// Mitsubishi GX Works2 project: R3R4R5 plc 20-08-2023_fr   PLC: Q03UDV

PROGRAM MAIN
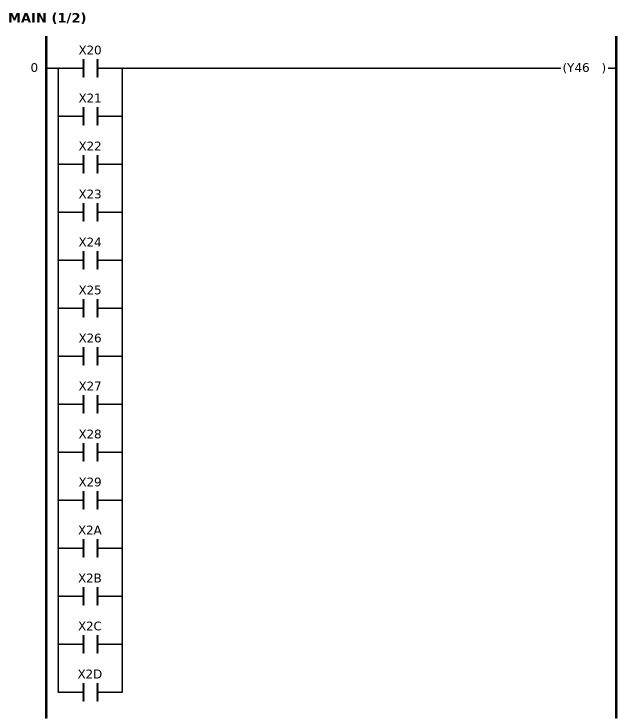
0     LD      X20
      OR      X21
      OR      X22
      OR      X23
      OR      X24
      OR      X25
      OR      X26
      OR      X27
      OR      X28
      OR      X29
      OR      X2A
      OR      X2B
      OR      X2C
      OR      X2D
      OUT     Y46
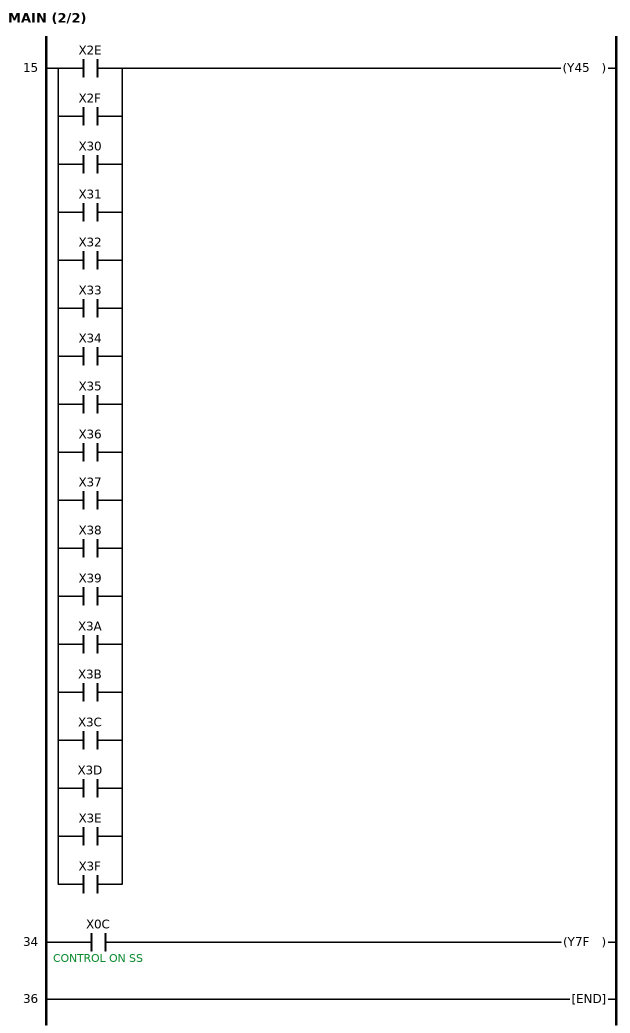
15    LD      X2E
      OR      X2F
      OR      X30
      OR      X31
      OR      X32
      OR      X33
      OR      X34
      OR      X35
      OR      X36
      OR      X37
      OR      X38
      OR      X39
      OR      X3A
      OR      X3B
      OR      X3C
      OR      X3D
      OR      X3E
      OR      X3F
      OUT     Y45
34    LD      X0C  ; CONTROL ON SS
      OUT     Y7F
36    END
END_PROGRAM

PROGRAM DEVICNET
0     END
END_PROGRAM

PROGRAM AUTO_PRG
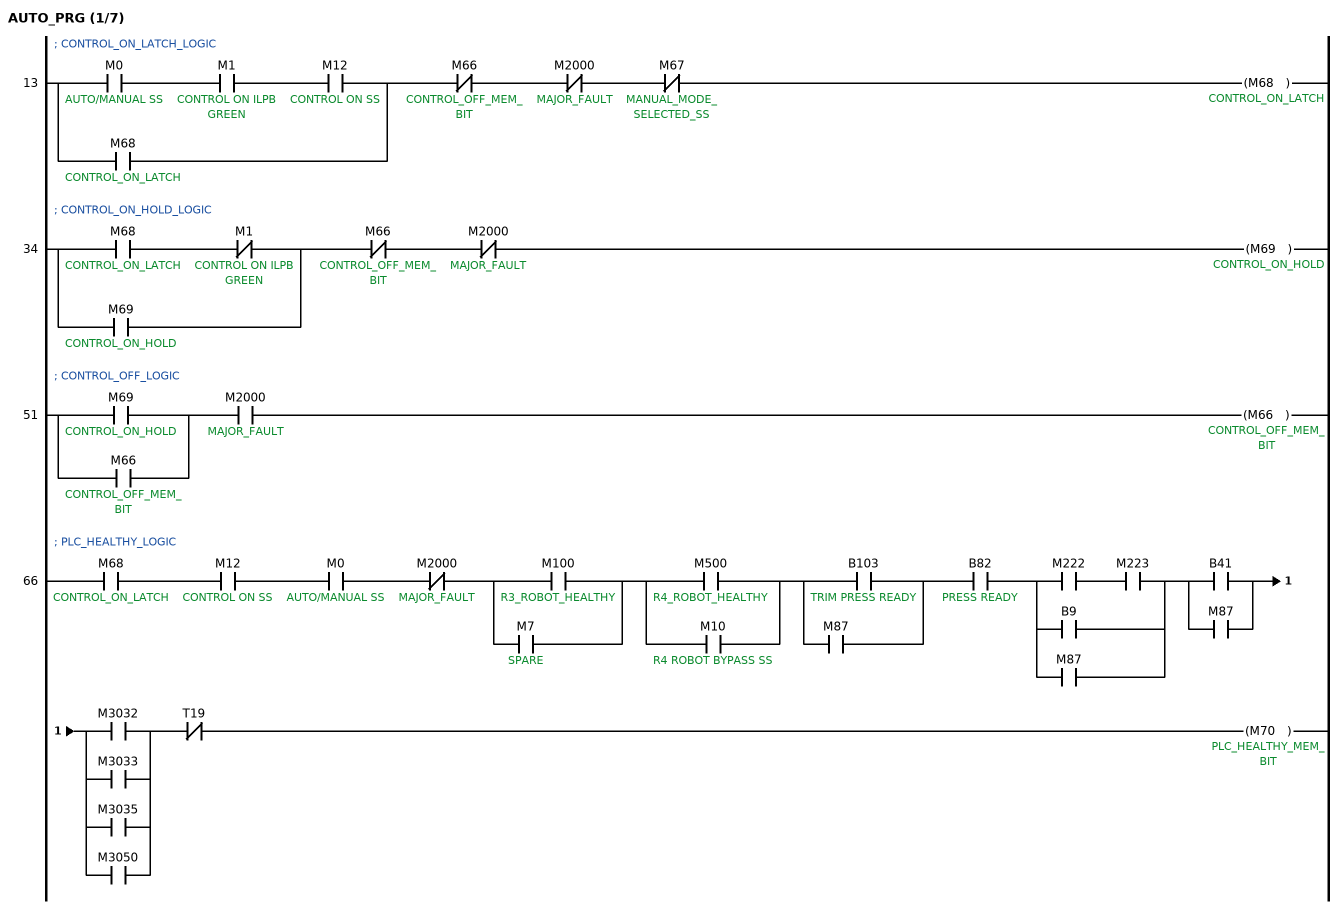
; CONTROL_ON_LATCH_LOGIC
13    LD      M0  ; AUTO/MANUAL SS
      AND     M1  ; CONTROL ON ILPB GREEN
      AND     M12  ; CONTROL ON SS
      OR      M68  ; CONTROL_ON_LATCH
      ANI     M66  ; CONTROL_OFF_MEM_BIT
      ANI     M2000  ; MAJOR_FAULT
      ANI     M67  ; MANUAL_MODE_SELECTED_SS
      OUT     M68  ; CONTROL_ON_LATCH
; CONTROL_ON_HOLD_LOGIC
34    LD      M68  ; CONTROL_ON_LATCH
      ANI     M1  ; CONTROL ON ILPB GREEN
      OR      M69  ; CONTROL_ON_HOLD
      ANI     M66  ; CONTROL_OFF_MEM_BIT
      ANI     M2000  ; MAJOR_FAULT
      OUT     M69  ; CONTROL_ON_HOLD
; CONTROL_OFF_LOGIC
51    LD      M69  ; CONTROL_ON_HOLD
      OR      M66  ; CONTROL_OFF_MEM_BIT
      AND     M2000  ; MAJOR_FAULT
      OUT     M66  ; CONTROL_OFF_MEM_BIT
; PLC_HEALTHY_LOGIC
66    LD      M68  ; CONTROL_ON_LATCH
      AND     M12  ; CONTROL ON SS
      AND     M0  ; AUTO/MANUAL SS
      ANI     M2000  ; MAJOR_FAULT
      LD      M100  ; R3_ROBOT_HEALTHY
      OR      M7  ; SPARE
      ANB
      LD      M500  ; R4_ROBOT_HEALTHY
      OR      M10  ; R4 ROBOT BYPASS SS
      ANB
      LD      B103  ; TRIM PRESS READY
      OR      M87
      ANB
      AND     B82  ; PRESS READY
      LD      M222
      AND     M223
      OR      B9
      OR      M87
      ANB
      LD      B41
      OR      M87
      ANB
      LD      M3032
      OR      M3033
      OR      M3035
      OR      M3050
      ANB
      ANI     T19
      OUT     M70  ; PLC_HEALTHY_MEM_BIT
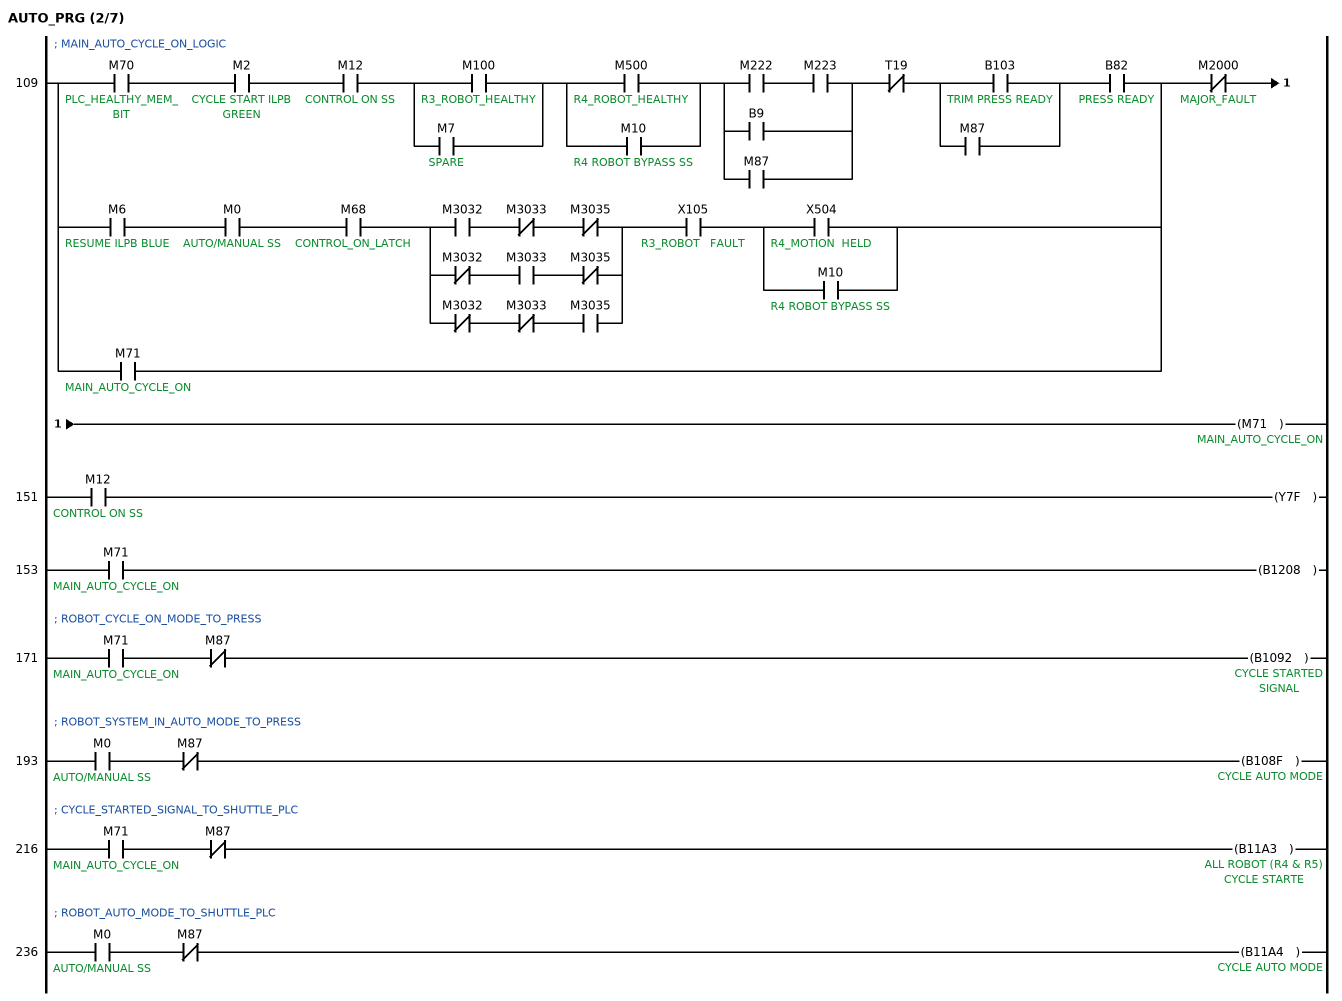
; MAIN_AUTO_CYCLE_ON_LOGIC
109   LD      M70  ; PLC_HEALTHY_MEM_BIT
      AND     M2  ; CYCLE START ILPB GREEN
      AND     M12  ; CONTROL ON SS
      LD      M100  ; R3_ROBOT_HEALTHY
      OR      M7  ; SPARE
      ANB
      LD      M500  ; R4_ROBOT_HEALTHY
      OR      M10  ; R4 ROBOT BYPASS SS
      ANB
      LD      M222
      AND     M223
      OR      B9
      OR      M87
      ANB
      ANI     T19
      LD      B103  ; TRIM PRESS READY
      OR      M87
      ANB
      AND     B82  ; PRESS READY
      LD      M6  ; RESUME ILPB BLUE
      AND     M0  ; AUTO/MANUAL SS
      AND     M68  ; CONTROL_ON_LATCH
      LD      M3032
      ANI     M3033
      ANI     M3035
      LDI     M3032
      AND     M3033
      ANI     M3035
      ORB
      LDI     M3032
      ANI     M3033
      AND     M3035
      ORB
      ANB
      AND     X105  ; R3_ROBOT   FAULT
      LD      X504  ; R4_MOTION  HELD
      OR      M10  ; R4 ROBOT BYPASS SS
      ANB
      ORB
      OR      M71  ; MAIN_AUTO_CYCLE_ON
      ANI     M2000  ; MAJOR_FAULT
      OUT     M71  ; MAIN_AUTO_CYCLE_ON
151   LD      M12  ; CONTROL ON SS
      OUT     Y7F
153   LD      M71  ; MAIN_AUTO_CYCLE_ON
      OUT     B1208
; ROBOT_CYCLE_ON_MODE_TO_PRESS
171   LD      M71  ; MAIN_AUTO_CYCLE_ON
      ANI     M87
      OUT     B1092  ; CYCLE STARTED SIGNAL
; ROBOT_SYSTEM_IN_AUTO_MODE_TO_PRESS
193   LD      M0  ; AUTO/MANUAL SS
      ANI     M87
      OUT     B108F  ; CYCLE AUTO MODE
; CYCLE_STARTED_SIGNAL_TO_SHUTTLE_PLC
216   LD      M71  ; MAIN_AUTO_CYCLE_ON
      ANI     M87
      OUT     B11A3  ; ALL ROBOT (R4 & R5) CYCLE STARTE
; ROBOT_AUTO_MODE_TO_SHUTTLE_PLC
236   LD      M0  ; AUTO/MANUAL SS
      ANI     M87
      OUT     B11A4  ; CYCLE AUTO MODE
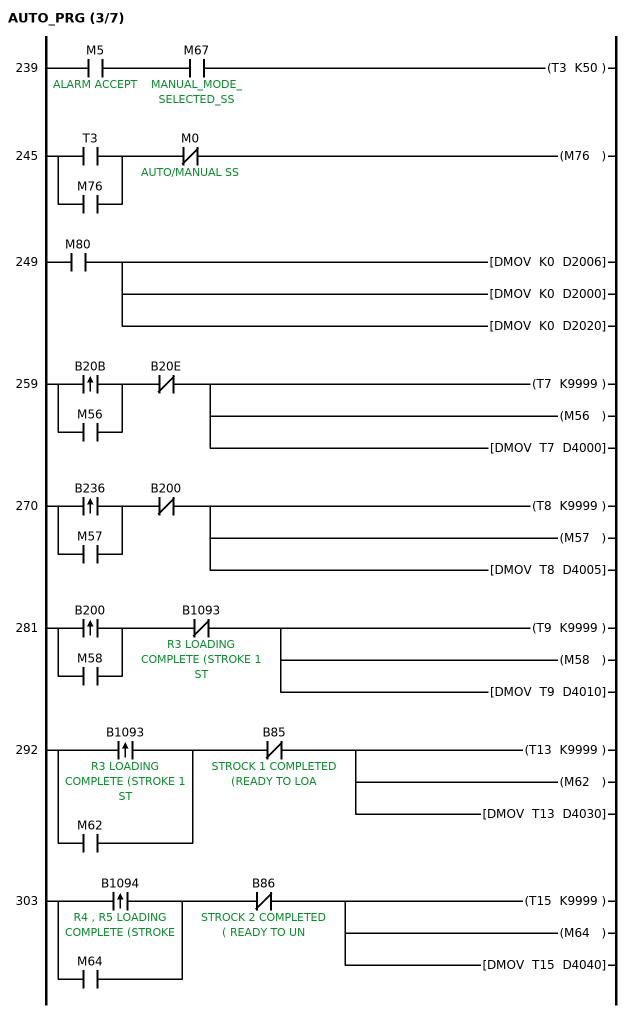
239   LD      M5  ; ALARM ACCEPT
      AND     M67  ; MANUAL_MODE_SELECTED_SS
      OUT     T3 K50
245   LD      T3
      OR      M76
      ANI     M0  ; AUTO/MANUAL SS
      OUT     M76
249   LD      M80
      DMOV    K0 D2006
      DMOV    K0 D2000
      DMOV    K0 D2020
259   LDP     B20B
      OR      M56
      ANI     B20E
      OUT     T7 K9999
      OUT     M56
      DMOV    T7 D4000
270   LDP     B236
      OR      M57
      ANI     B200
      OUT     T8 K9999
      OUT     M57
      DMOV    T8 D4005
281   LDP     B200
      OR      M58
      ANI     B1093  ; R3 LOADING COMPLETE (STROKE 1 ST
      OUT     T9 K9999
      OUT     M58
      DMOV    T9 D4010
292   LDP     B1093  ; R3 LOADING COMPLETE (STROKE 1 ST
      OR      M62
      ANI     B85  ; STROCK 1 COMPLETED (READY TO LOA
      OUT     T13 K9999
      OUT     M62
      DMOV    T13 D4030
303   LDP     B1094  ; R4 , R5 LOADING COMPLETE (STROKE
      OR      M64
      ANI     B86  ; STROCK 2 COMPLETED ( READY TO UN
      OUT     T15 K9999
      OUT     M64
      DMOV    T15 D4040
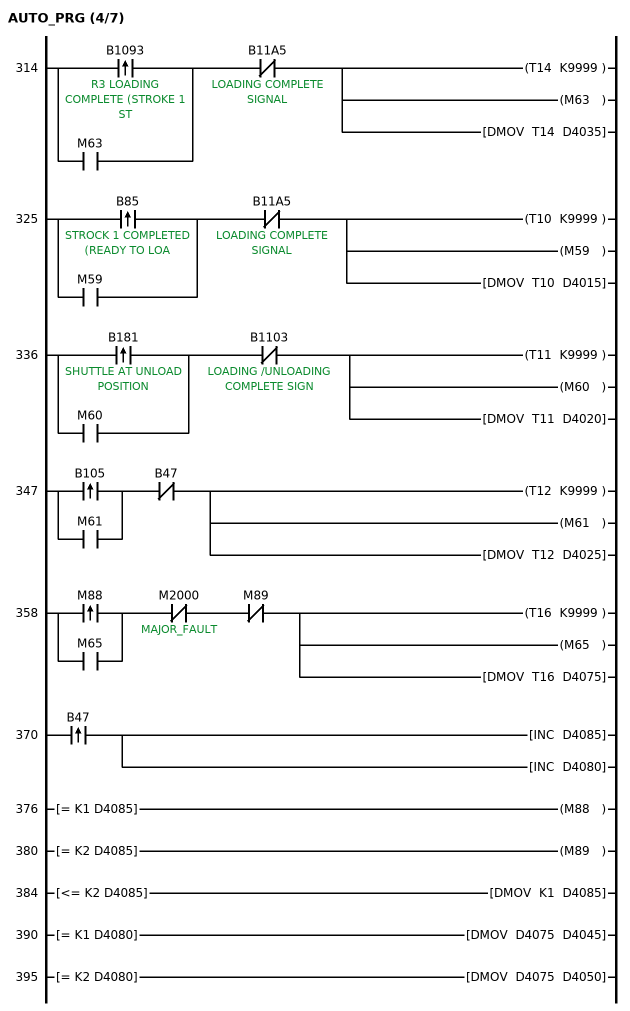
314   LDP     B1093  ; R3 LOADING COMPLETE (STROKE 1 ST
      OR      M63
      ANI     B11A5  ; LOADING COMPLETE SIGNAL
      OUT     T14 K9999
      OUT     M63
      DMOV    T14 D4035
325   LDP     B85  ; STROCK 1 COMPLETED (READY TO LOA
      OR      M59
      ANI     B11A5  ; LOADING COMPLETE SIGNAL
      OUT     T10 K9999
      OUT     M59
      DMOV    T10 D4015
336   LDP     B181  ; SHUTTLE AT UNLOAD POSITION
      OR      M60
      ANI     B1103  ; LOADING /UNLOADING COMPLETE SIGN
      OUT     T11 K9999
      OUT     M60
      DMOV    T11 D4020
347   LDP     B105
      OR      M61
      ANI     B47
      OUT     T12 K9999
      OUT     M61
      DMOV    T12 D4025
358   LDP     M88
      OR      M65
      ANI     M2000  ; MAJOR_FAULT
      ANI     M89
      OUT     T16 K9999
      OUT     M65
      DMOV    T16 D4075
370   LDP     B47
      INC     D4085
      INC     D4080
376   LD=     K1 D4085
      OUT     M88
380   LD=     K2 D4085
      OUT     M89
384   LD<=    K2 D4085
      DMOV    K1 D4085
390   LD=     K1 D4080
      DMOV    D4075 D4045
395   LD=     K2 D4080
      DMOV    D4075 D4050
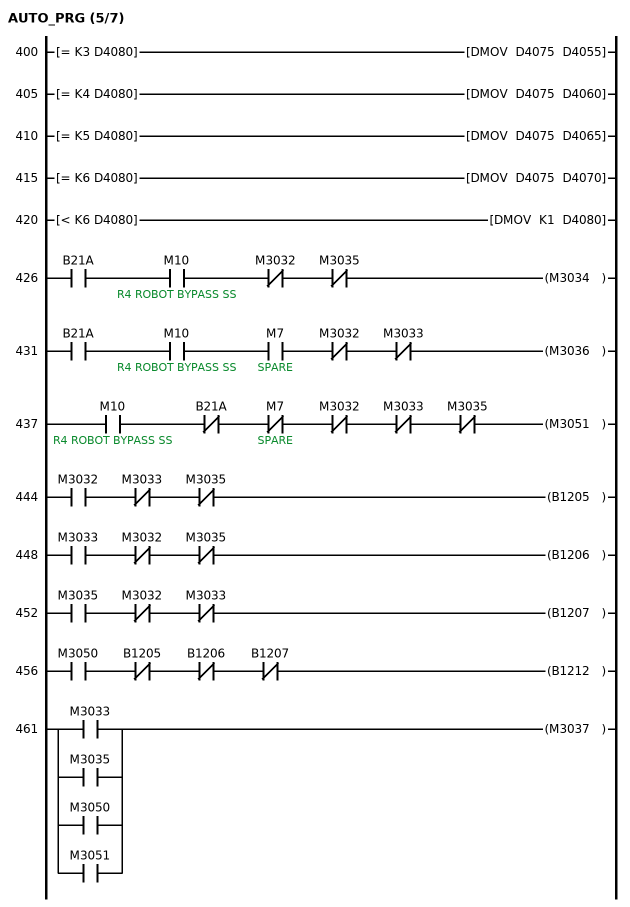
400   LD=     K3 D4080
      DMOV    D4075 D4055
405   LD=     K4 D4080
      DMOV    D4075 D4060
410   LD=     K5 D4080
      DMOV    D4075 D4065
415   LD=     K6 D4080
      DMOV    D4075 D4070
420   LD<     K6 D4080
      DMOV    K1 D4080
426   LD      B21A
      AND     M10  ; R4 ROBOT BYPASS SS
      ANI     M3032
      ANI     M3035
      OUT     M3034
431   LD      B21A
      AND     M10  ; R4 ROBOT BYPASS SS
      AND     M7  ; SPARE
      ANI     M3032
      ANI     M3033
      OUT     M3036
437   LD      M10  ; R4 ROBOT BYPASS SS
      ANI     B21A
      ANI     M7  ; SPARE
      ANI     M3032
      ANI     M3033
      ANI     M3035
      OUT     M3051
444   LD      M3032
      ANI     M3033
      ANI     M3035
      OUT     B1205
448   LD      M3033
      ANI     M3032
      ANI     M3035
      OUT     B1206
452   LD      M3035
      ANI     M3032
      ANI     M3033
      OUT     B1207
456   LD      M3050
      ANI     B1205
      ANI     B1206
      ANI     B1207
      OUT     B1212
461   LD      M3033
      OR      M3035
      OR      M3050
      OR      M3051
      OUT     M3037
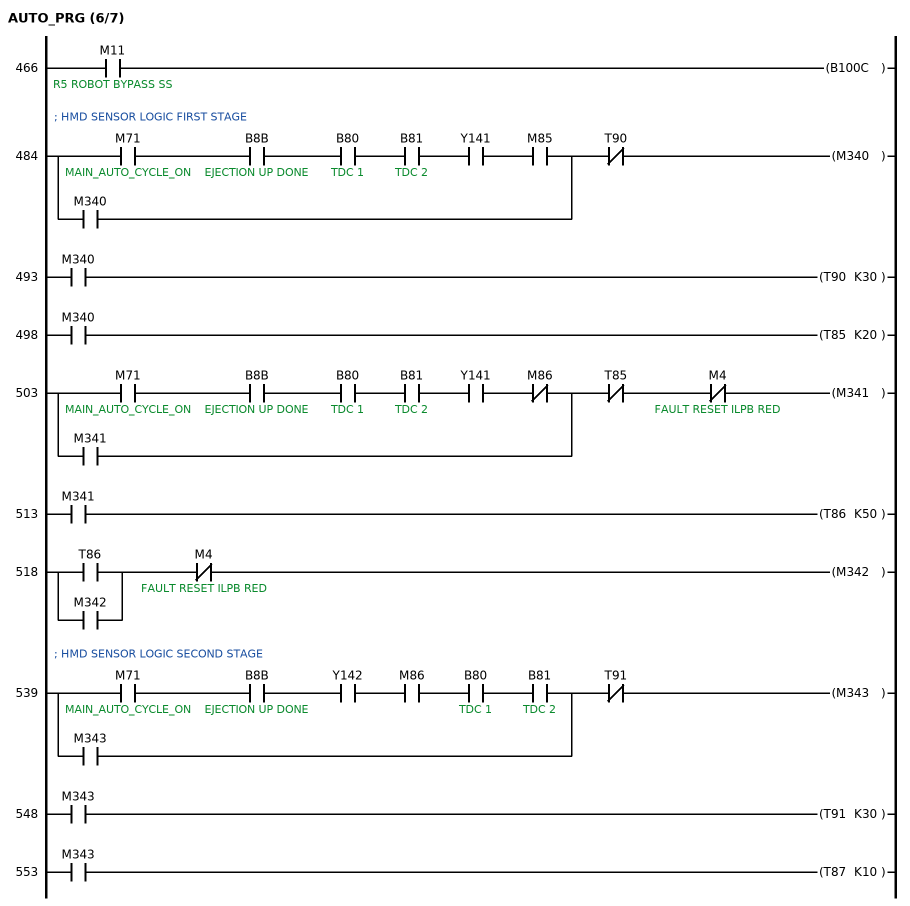
466   LD      M11  ; R5 ROBOT BYPASS SS
      OUT     B100C
; HMD SENSOR LOGIC FIRST STAGE
484   LD      M71  ; MAIN_AUTO_CYCLE_ON
      AND     B8B  ; EJECTION UP DONE
      AND     B80  ; TDC 1
      AND     B81  ; TDC 2
      AND     Y141
      AND     M85
      OR      M340
      ANI     T90
      OUT     M340
493   LD      M340
      OUT     T90 K30
498   LD      M340
      OUT     T85 K20
503   LD      M71  ; MAIN_AUTO_CYCLE_ON
      AND     B8B  ; EJECTION UP DONE
      AND     B80  ; TDC 1
      AND     B81  ; TDC 2
      AND     Y141
      ANI     M86
      OR      M341
      ANI     T85
      ANI     M4  ; FAULT RESET ILPB RED
      OUT     M341
513   LD      M341
      OUT     T86 K50
518   LD      T86
      OR      M342
      ANI     M4  ; FAULT RESET ILPB RED
      OUT     M342
; HMD SENSOR LOGIC SECOND STAGE
539   LD      M71  ; MAIN_AUTO_CYCLE_ON
      AND     B8B  ; EJECTION UP DONE
      AND     Y142
      AND     M86
      AND     B80  ; TDC 1
      AND     B81  ; TDC 2
      OR      M343
      ANI     T91
      OUT     M343
548   LD      M343
      OUT     T91 K30
553   LD      M343
      OUT     T87 K10
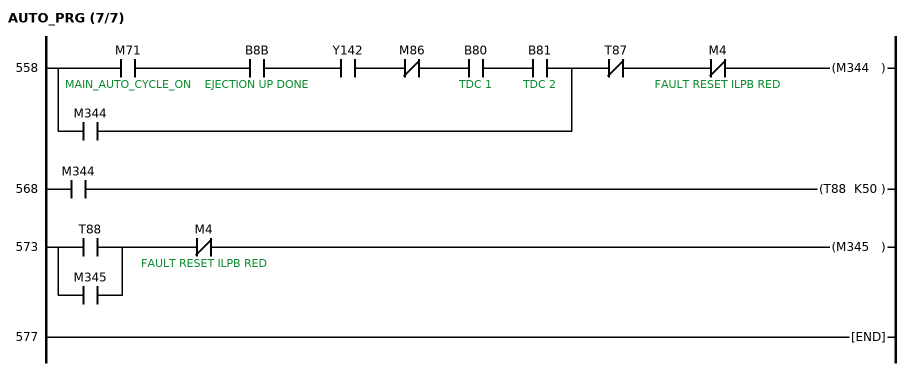
558   LD      M71  ; MAIN_AUTO_CYCLE_ON
      AND     B8B  ; EJECTION UP DONE
      AND     Y142
      ANI     M86
      AND     B80  ; TDC 1
      AND     B81  ; TDC 2
      OR      M344
      ANI     T87
      ANI     M4  ; FAULT RESET ILPB RED
      OUT     M344
568   LD      M344
      OUT     T88 K50
573   LD      T88
      OR      M345
      ANI     M4  ; FAULT RESET ILPB RED
      OUT     M345
577   END
END_PROGRAM

PROGRAM CC_LINK
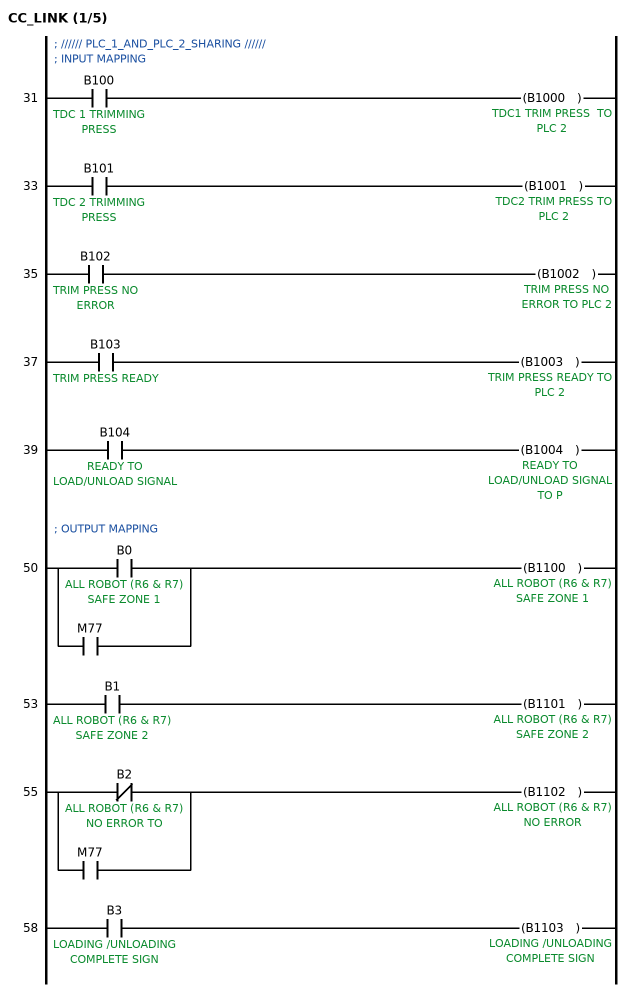
; ////// PLC_1_AND_PLC_2_SHARING //////
; 
; INPUT MAPPING
31    LD      B100  ; TDC 1 TRIMMING PRESS
      OUT     B1000  ; TDC1 TRIM PRESS  TO PLC 2
33    LD      B101  ; TDC 2 TRIMMING PRESS
      OUT     B1001  ; TDC2 TRIM PRESS TO PLC 2
35    LD      B102  ; TRIM PRESS NO ERROR
      OUT     B1002  ; TRIM PRESS NO ERROR TO PLC 2
37    LD      B103  ; TRIM PRESS READY
      OUT     B1003  ; TRIM PRESS READY TO PLC 2
39    LD      B104  ; READY TO LOAD/UNLOAD SIGNAL
      OUT     B1004  ; READY TO LOAD/UNLOAD SIGNAL TO P
; OUTPUT MAPPING
50    LD      B0  ; ALL ROBOT (R6 & R7) SAFE ZONE 1
      OR      M77
      OUT     B1100  ; ALL ROBOT (R6 & R7) SAFE ZONE 1
53    LD      B1  ; ALL ROBOT (R6 & R7) SAFE ZONE 2
      OUT     B1101  ; ALL ROBOT (R6 & R7) SAFE ZONE 2
55    LDI     B2  ; ALL ROBOT (R6 & R7) NO ERROR TO
      OR      M77
      OUT     B1102  ; ALL ROBOT (R6 & R7) NO ERROR
58    LD      B3  ; LOADING /UNLOADING COMPLETE SIGN
      OUT     B1103  ; LOADING /UNLOADING COMPLETE SIGN
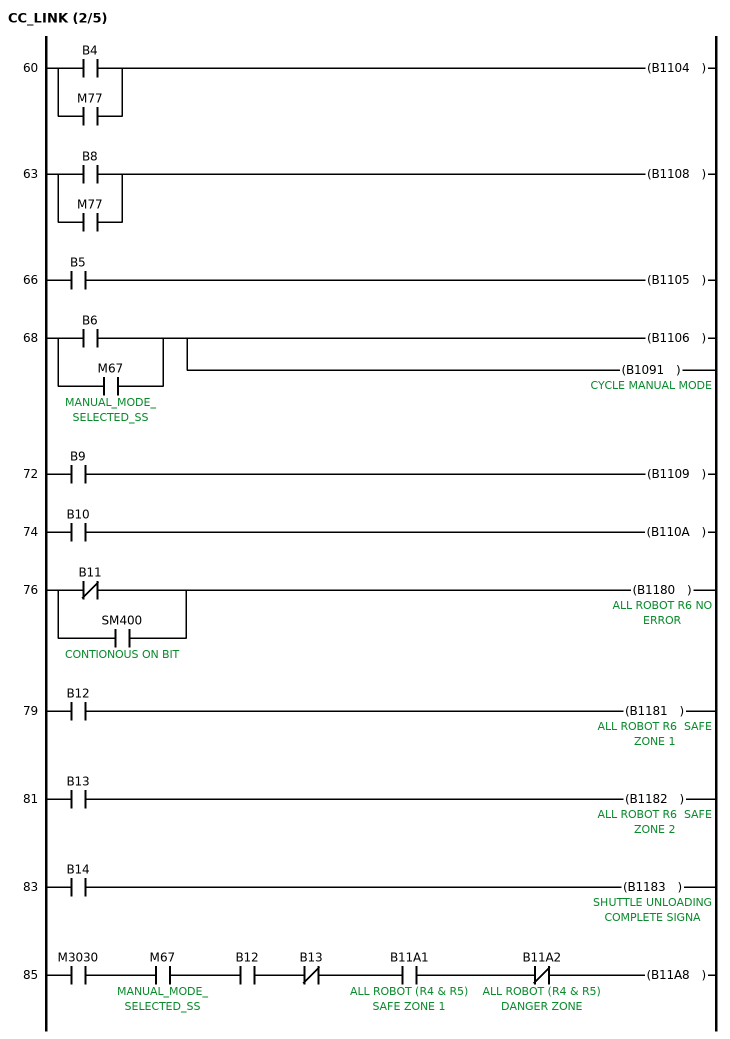
60    LD      B4
      OR      M77
      OUT     B1104
63    LD      B8
      OR      M77
      OUT     B1108
66    LD      B5
      OUT     B1105
68    LD      B6
      OR      M67  ; MANUAL_MODE_SELECTED_SS
      OUT     B1106
      OUT     B1091  ; CYCLE MANUAL MODE
72    LD      B9
      OUT     B1109
74    LD      B10
      OUT     B110A
76    LDI     B11
      OR      SM400  ; CONTIONOUS ON BIT
      OUT     B1180  ; ALL ROBOT R6 NO ERROR
79    LD      B12
      OUT     B1181  ; ALL ROBOT R6  SAFE ZONE 1
81    LD      B13
      OUT     B1182  ; ALL ROBOT R6  SAFE ZONE 2
83    LD      B14
      OUT     B1183  ; SHUTTLE UNLOADING COMPLETE SIGNA
85    LD      M3030
      AND     M67  ; MANUAL_MODE_SELECTED_SS
      AND     B12
      ANI     B13
      AND     B11A1  ; ALL ROBOT (R4 & R5) SAFE ZONE 1
      ANI     B11A2  ; ALL ROBOT (R4 & R5) DANGER ZONE
      OUT     B11A8
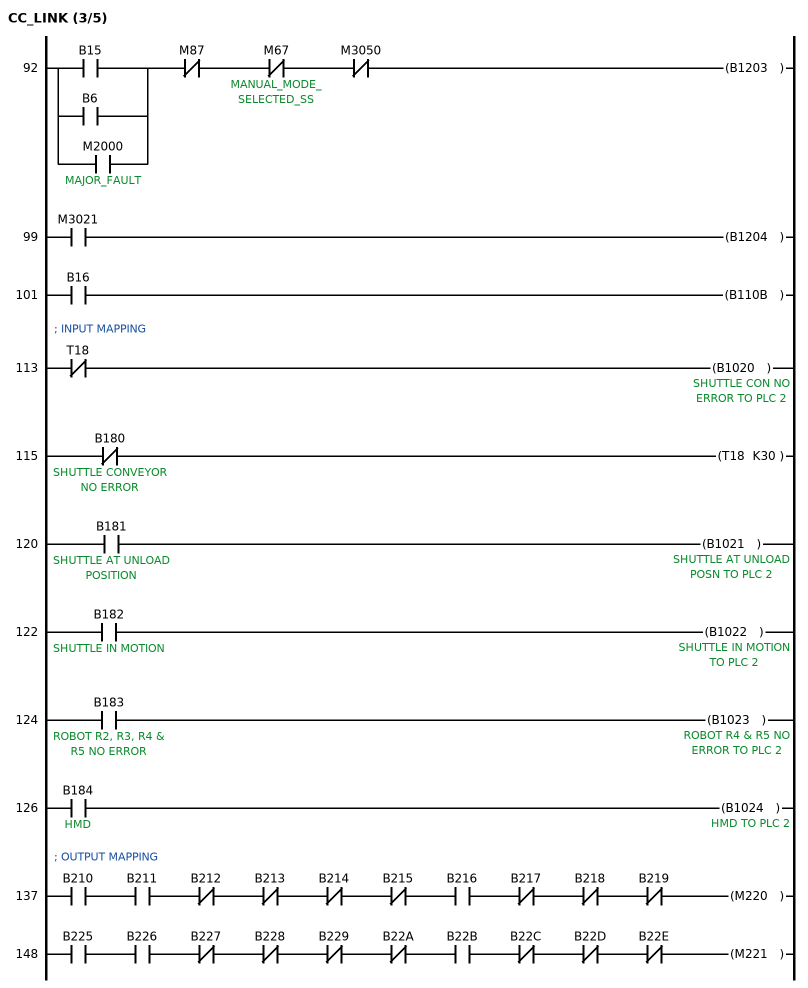
92    LD      B15
      OR      B6
      OR      M2000  ; MAJOR_FAULT
      ANI     M87
      ANI     M67  ; MANUAL_MODE_SELECTED_SS
      ANI     M3050
      OUT     B1203
99    LD      M3021
      OUT     B1204
101   LD      B16
      OUT     B110B
; 
; INPUT MAPPING
113   LDI     T18
      OUT     B1020  ; SHUTTLE CON NO ERROR TO PLC 2
115   LDI     B180  ; SHUTTLE CONVEYOR NO ERROR
      OUT     T18 K30
120   LD      B181  ; SHUTTLE AT UNLOAD POSITION
      OUT     B1021  ; SHUTTLE AT UNLOAD POSN TO PLC 2
122   LD      B182  ; SHUTTLE IN MOTION
      OUT     B1022  ; SHUTTLE IN MOTION TO PLC 2
124   LD      B183  ; ROBOT R2, R3, R4 & R5 NO ERROR
      OUT     B1023  ; ROBOT R4 & R5 NO ERROR TO PLC 2
126   LD      B184  ; HMD
      OUT     B1024  ; HMD TO PLC 2
; OUTPUT MAPPING
137   LD      B210
      AND     B211
      ANI     B212
      ANI     B213
      ANI     B214
      ANI     B215
      AND     B216
      ANI     B217
      ANI     B218
      ANI     B219
      OUT     M220
148   LD      B225
      AND     B226
      ANI     B227
      ANI     B228
      ANI     B229
      ANI     B22A
      AND     B22B
      ANI     B22C
      ANI     B22D
      ANI     B22E
      OUT     M221
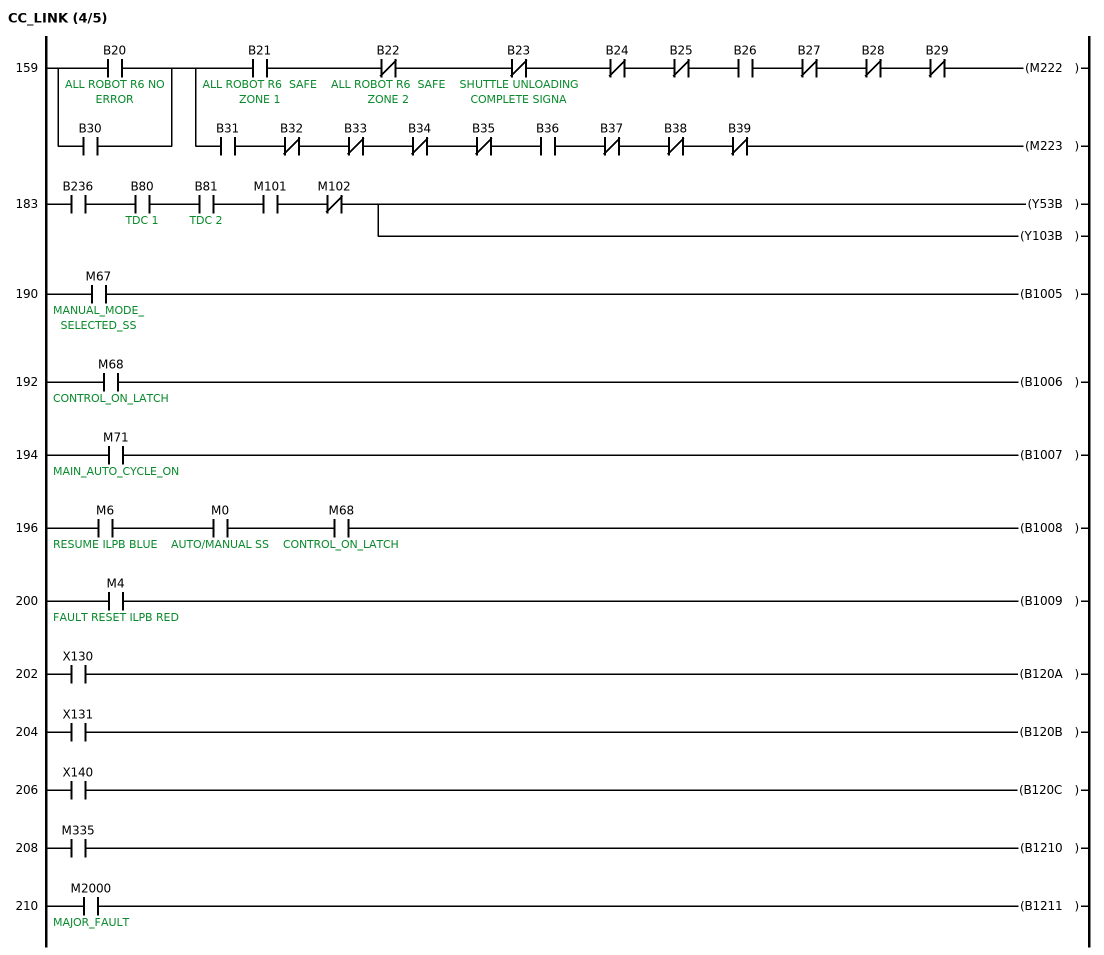
159   LD      B20  ; ALL ROBOT R6 NO ERROR
      OR      B30
      MPS
      AND     B21  ; ALL ROBOT R6  SAFE ZONE 1
      ANI     B22  ; ALL ROBOT R6  SAFE ZONE 2
      ANI     B23  ; SHUTTLE UNLOADING COMPLETE SIGNA
      ANI     B24
      ANI     B25
      AND     B26
      ANI     B27
      ANI     B28
      ANI     B29
      OUT     M222
      MPP
      AND     B31
      ANI     B32
      ANI     B33
      ANI     B34
      ANI     B35
      AND     B36
      ANI     B37
      ANI     B38
      ANI     B39
      OUT     M223
183   LD      B236
      AND     B80  ; TDC 1
      AND     B81  ; TDC 2
      AND     M101
      ANI     M102
      OUT     Y53B
      OUT     Y103B
190   LD      M67  ; MANUAL_MODE_SELECTED_SS
      OUT     B1005
192   LD      M68  ; CONTROL_ON_LATCH
      OUT     B1006
194   LD      M71  ; MAIN_AUTO_CYCLE_ON
      OUT     B1007
196   LD      M6  ; RESUME ILPB BLUE
      AND     M0  ; AUTO/MANUAL SS
      AND     M68  ; CONTROL_ON_LATCH
      OUT     B1008
200   LD      M4  ; FAULT RESET ILPB RED
      OUT     B1009
202   LD      X130
      OUT     B120A
204   LD      X131
      OUT     B120B
206   LD      X140
      OUT     B120C
208   LD      M335
      OUT     B1210
210   LD      M2000  ; MAJOR_FAULT
      OUT     B1211
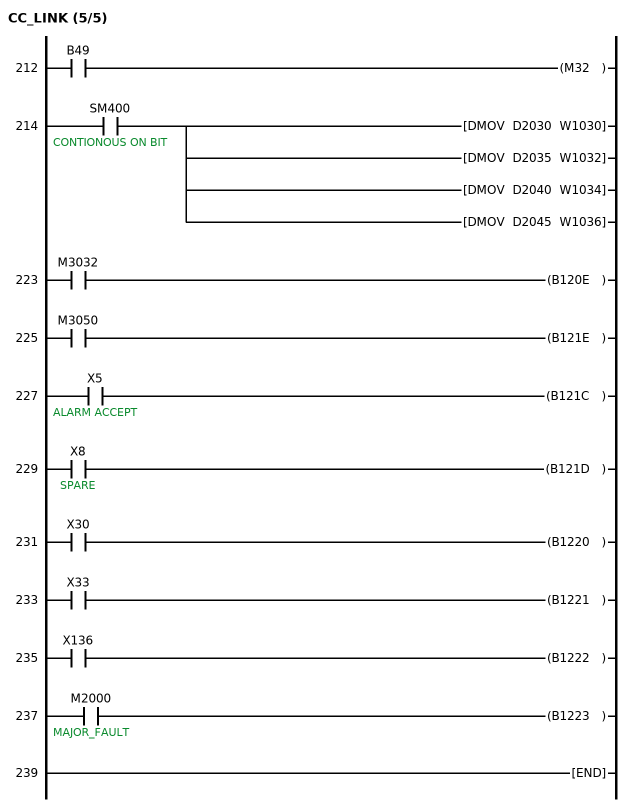
212   LD      B49
      OUT     M32
214   LD      SM400  ; CONTIONOUS ON BIT
      DMOV    D2030 W1030
      DMOV    D2035 W1032
      DMOV    D2040 W1034
      DMOV    D2045 W1036
223   LD      M3032
      OUT     B120E
225   LD      M3050
      OUT     B121E
227   LD      X5  ; ALARM ACCEPT
      OUT     B121C
229   LD      X8  ; SPARE
      OUT     B121D
231   LD      X30
      OUT     B1220
233   LD      X33
      OUT     B1221
235   LD      X136
      OUT     B1222
237   LD      M2000  ; MAJOR_FAULT
      OUT     B1223
239   END
END_PROGRAM

PROGRAM DEVICE_N
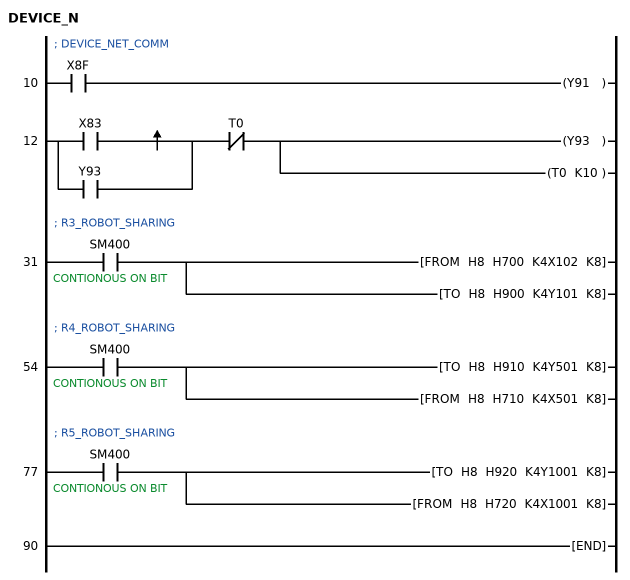
; DEVICE_NET_COMM
10    LD      X8F
      OUT     Y91
12    LD      X83
      MEP
      OR      Y93
      ANI     T0
      OUT     Y93
      OUT     T0 K10
; R3_ROBOT_SHARING
31    LD      SM400  ; CONTIONOUS ON BIT
      FROM    H8 H700 K4X102 K8  ; R3_PROGRAM RUNNING
      TO      H8 H900 K4Y101 K8  ; R3_HOLD TO ROBOT
; R4_ROBOT_SHARING
54    LD      SM400  ; CONTIONOUS ON BIT
      TO      H8 H910 K4Y501 K8  ; R4_HOLD TO ROBOT
      FROM    H8 H710 K4X501 K8  ; R4_SYSTEM  READY
; R5_ROBOT_SHARING
77    LD      SM400  ; CONTIONOUS ON BIT
      TO      H8 H920 K4Y1001 K8  ; R5_HOLD TO ROBOT
      FROM    H8 H720 K4X1001 K8  ; R5_SYSTEM  READY
90    END
END_PROGRAM

PROGRAM FAULT
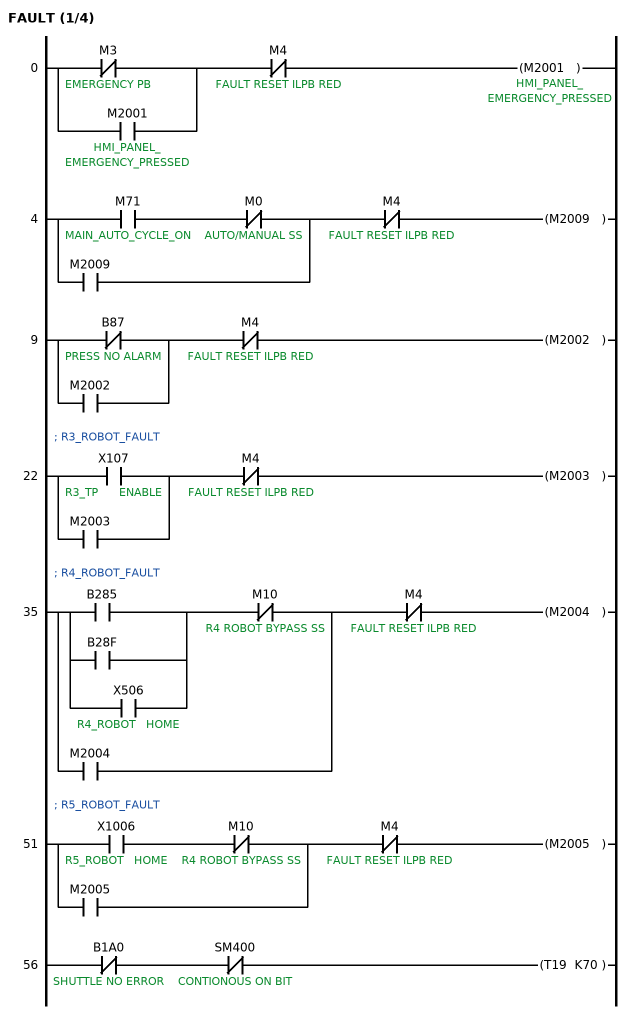
0     LDI     M3  ; EMERGENCY PB
      OR      M2001  ; HMI_PANEL_EMERGENCY_PRESSED
      ANI     M4  ; FAULT RESET ILPB RED
      OUT     M2001  ; HMI_PANEL_EMERGENCY_PRESSED
4     LD      M71  ; MAIN_AUTO_CYCLE_ON
      ANI     M0  ; AUTO/MANUAL SS
      OR      M2009
      ANI     M4  ; FAULT RESET ILPB RED
      OUT     M2009
9     LDI     B87  ; PRESS NO ALARM
      OR      M2002
      ANI     M4  ; FAULT RESET ILPB RED
      OUT     M2002
; R3_ROBOT_FAULT
22    LD      X107  ; R3_TP      ENABLE
      OR      M2003
      ANI     M4  ; FAULT RESET ILPB RED
      OUT     M2003
; R4_ROBOT_FAULT
35    LD      B285
      OR      B28F
      OR      X506  ; R4_ROBOT   HOME
      ANI     M10  ; R4 ROBOT BYPASS SS
      OR      M2004
      ANI     M4  ; FAULT RESET ILPB RED
      OUT     M2004
; R5_ROBOT_FAULT
51    LD      X1006  ; R5_ROBOT   HOME
      ANI     M10  ; R4 ROBOT BYPASS SS
      OR      M2005
      ANI     M4  ; FAULT RESET ILPB RED
      OUT     M2005
56    LDI     B1A0  ; SHUTTLE NO ERROR
      ANI     SM400  ; CONTIONOUS ON BIT
      OUT     T19 K70
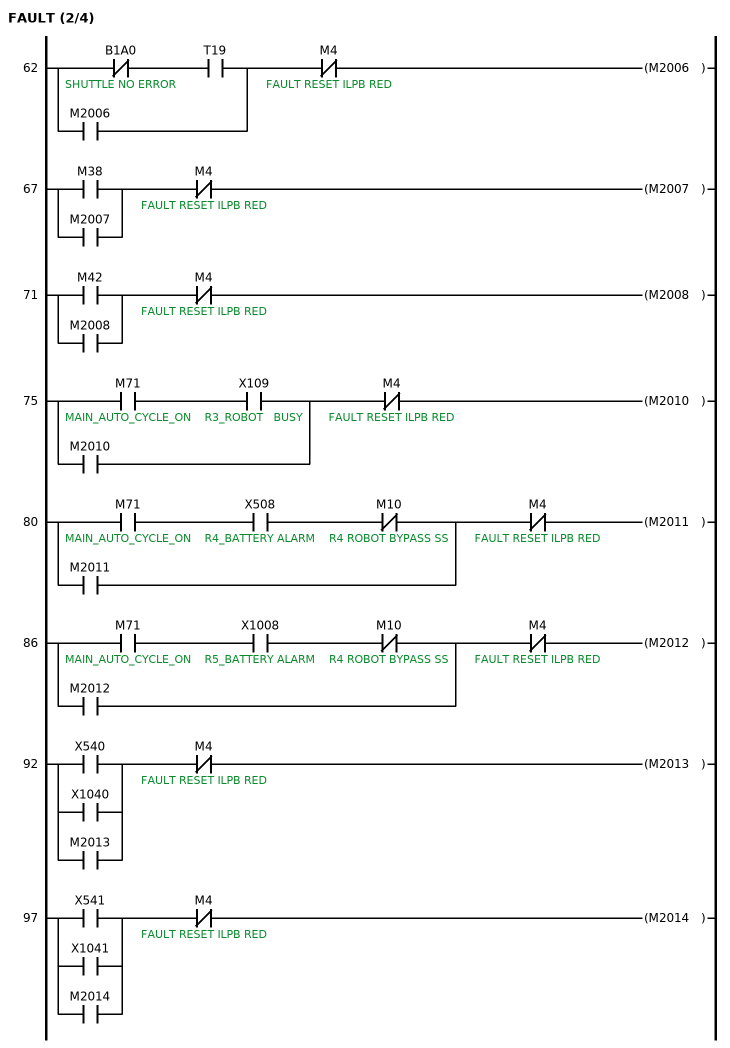
62    LDI     B1A0  ; SHUTTLE NO ERROR
      AND     T19
      OR      M2006
      ANI     M4  ; FAULT RESET ILPB RED
      OUT     M2006
67    LD      M38
      OR      M2007
      ANI     M4  ; FAULT RESET ILPB RED
      OUT     M2007
71    LD      M42
      OR      M2008
      ANI     M4  ; FAULT RESET ILPB RED
      OUT     M2008
75    LD      M71  ; MAIN_AUTO_CYCLE_ON
      AND     X109  ; R3_ROBOT   BUSY
      OR      M2010
      ANI     M4  ; FAULT RESET ILPB RED
      OUT     M2010
80    LD      M71  ; MAIN_AUTO_CYCLE_ON
      AND     X508  ; R4_BATTERY ALARM
      ANI     M10  ; R4 ROBOT BYPASS SS
      OR      M2011
      ANI     M4  ; FAULT RESET ILPB RED
      OUT     M2011
86    LD      M71  ; MAIN_AUTO_CYCLE_ON
      AND     X1008  ; R5_BATTERY ALARM
      ANI     M10  ; R4 ROBOT BYPASS SS
      OR      M2012
      ANI     M4  ; FAULT RESET ILPB RED
      OUT     M2012
92    LD      X540
      OR      X1040
      OR      M2013
      ANI     M4  ; FAULT RESET ILPB RED
      OUT     M2013
97    LD      X541
      OR      X1041
      OR      M2014
      ANI     M4  ; FAULT RESET ILPB RED
      OUT     M2014
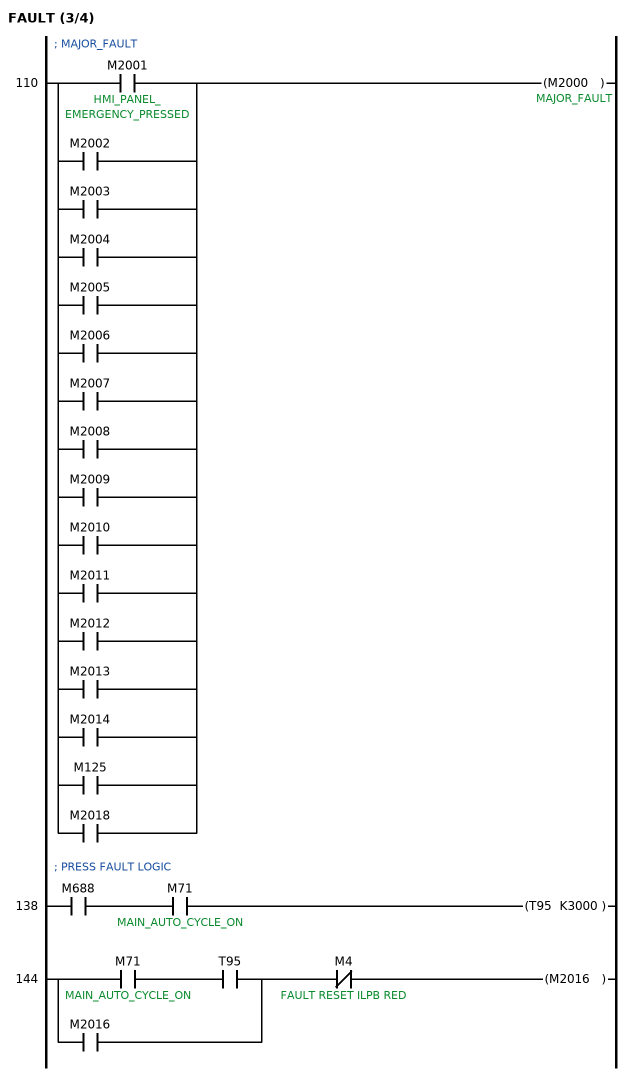
; MAJOR_FAULT
110   LD      M2001  ; HMI_PANEL_EMERGENCY_PRESSED
      OR      M2002
      OR      M2003
      OR      M2004
      OR      M2005
      OR      M2006
      OR      M2007
      OR      M2008
      OR      M2009
      OR      M2010
      OR      M2011
      OR      M2012
      OR      M2013
      OR      M2014
      OR      M125
      OR      M2018
      OUT     M2000  ; MAJOR_FAULT
; PRESS FAULT LOGIC
138   LD      M688
      AND     M71  ; MAIN_AUTO_CYCLE_ON
      OUT     T95 K3000
144   LD      M71  ; MAIN_AUTO_CYCLE_ON
      AND     T95
      OR      M2016
      ANI     M4  ; FAULT RESET ILPB RED
      OUT     M2016
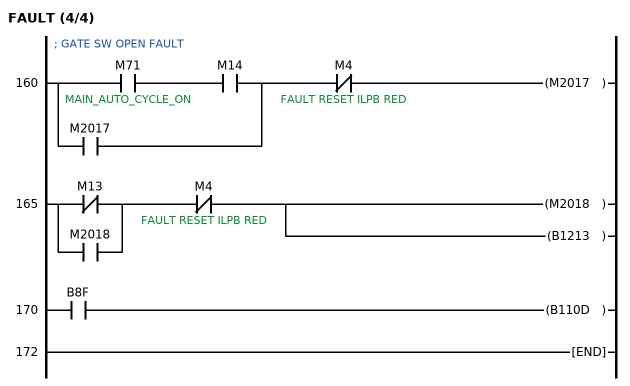
; GATE SW OPEN FAULT
160   LD      M71  ; MAIN_AUTO_CYCLE_ON
      AND     M14
      OR      M2017
      ANI     M4  ; FAULT RESET ILPB RED
      OUT     M2017
165   LDI     M13
      OR      M2018
      ANI     M4  ; FAULT RESET ILPB RED
      OUT     M2018
      OUT     B1213
170   LD      B8F
      OUT     B110D
172   END
END_PROGRAM

PROGRAM INPUT_MA
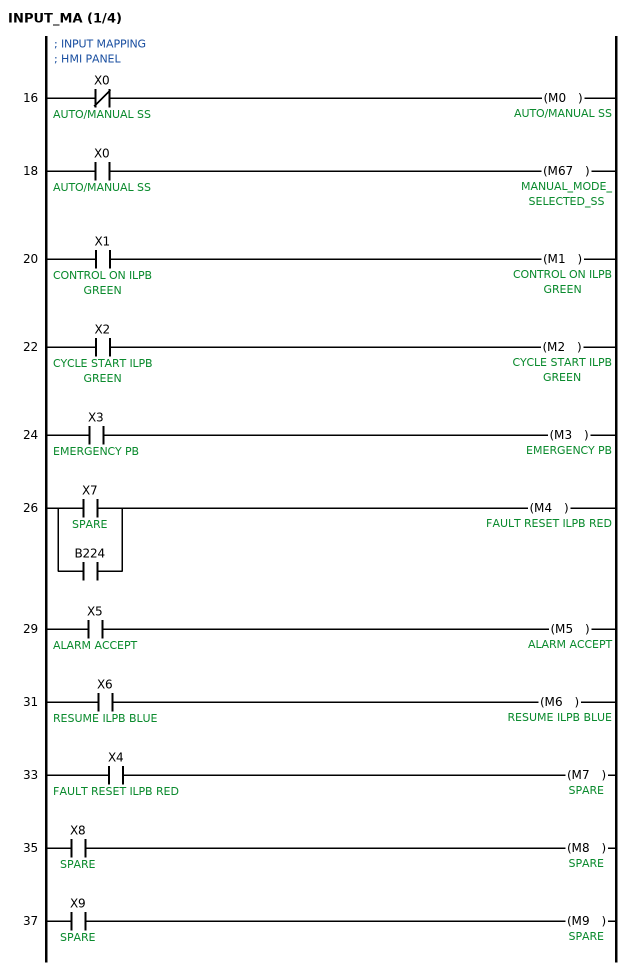
; INPUT MAPPING
; HMI PANEL
16    LDI     X0  ; AUTO/MANUAL SS
      OUT     M0  ; AUTO/MANUAL SS
18    LD      X0  ; AUTO/MANUAL SS
      OUT     M67  ; MANUAL_MODE_SELECTED_SS
20    LD      X1  ; CONTROL ON ILPB GREEN
      OUT     M1  ; CONTROL ON ILPB GREEN
22    LD      X2  ; CYCLE START ILPB GREEN
      OUT     M2  ; CYCLE START ILPB GREEN
24    LD      X3  ; EMERGENCY PB
      OUT     M3  ; EMERGENCY PB
26    LD      X7  ; SPARE
      OR      B224
      OUT     M4  ; FAULT RESET ILPB RED
29    LD      X5  ; ALARM ACCEPT
      OUT     M5  ; ALARM ACCEPT
31    LD      X6  ; RESUME ILPB BLUE
      OUT     M6  ; RESUME ILPB BLUE
33    LD      X4  ; FAULT RESET ILPB RED
      OUT     M7  ; SPARE
35    LD      X8  ; SPARE
      OUT     M8  ; SPARE
37    LD      X9  ; SPARE
      OUT     M9  ; SPARE
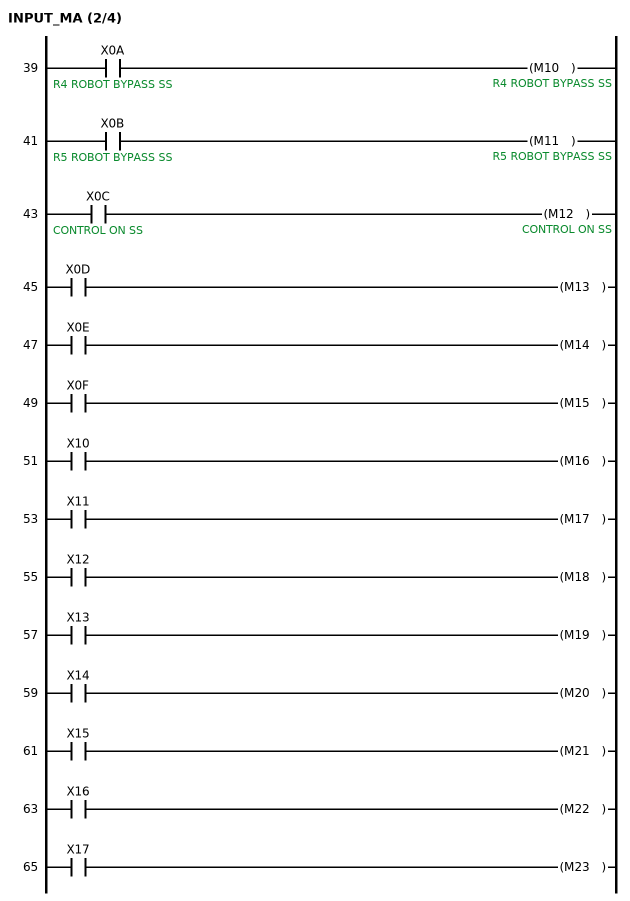
39    LD      X0A  ; R4 ROBOT BYPASS SS
      OUT     M10  ; R4 ROBOT BYPASS SS
41    LD      X0B  ; R5 ROBOT BYPASS SS
      OUT     M11  ; R5 ROBOT BYPASS SS
43    LD      X0C  ; CONTROL ON SS
      OUT     M12  ; CONTROL ON SS
45    LD      X0D
      OUT     M13
47    LD      X0E
      OUT     M14
49    LD      X0F
      OUT     M15
51    LD      X10
      OUT     M16
53    LD      X11
      OUT     M17
55    LD      X12
      OUT     M18
57    LD      X13
      OUT     M19
59    LD      X14
      OUT     M20
61    LD      X15
      OUT     M21
63    LD      X16
      OUT     M22
65    LD      X17
      OUT     M23
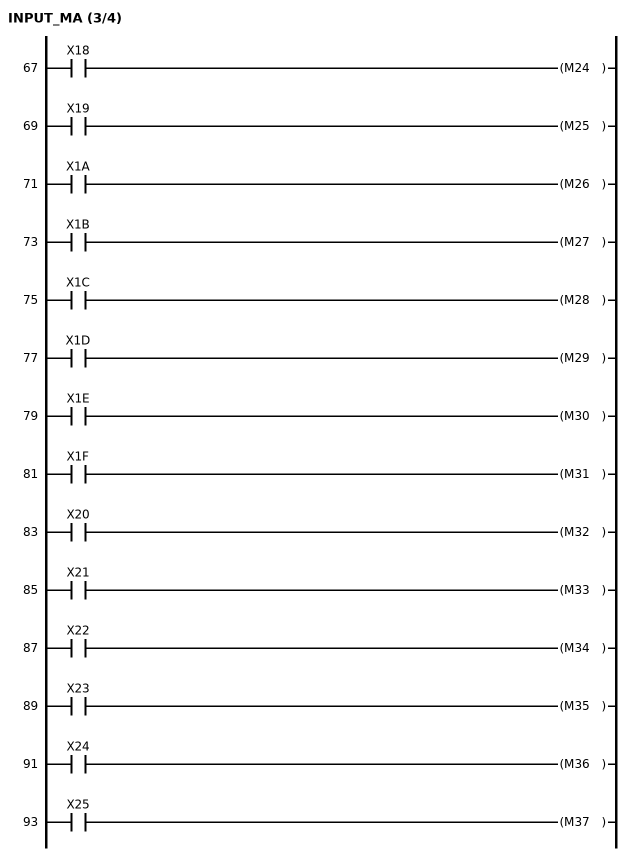
67    LD      X18
      OUT     M24
69    LD      X19
      OUT     M25
71    LD      X1A
      OUT     M26
73    LD      X1B
      OUT     M27
75    LD      X1C
      OUT     M28
77    LD      X1D
      OUT     M29
79    LD      X1E
      OUT     M30
81    LD      X1F
      OUT     M31
83    LD      X20
      OUT     M32
85    LD      X21
      OUT     M33
87    LD      X22
      OUT     M34
89    LD      X23
      OUT     M35
91    LD      X24
      OUT     M36
93    LD      X25
      OUT     M37
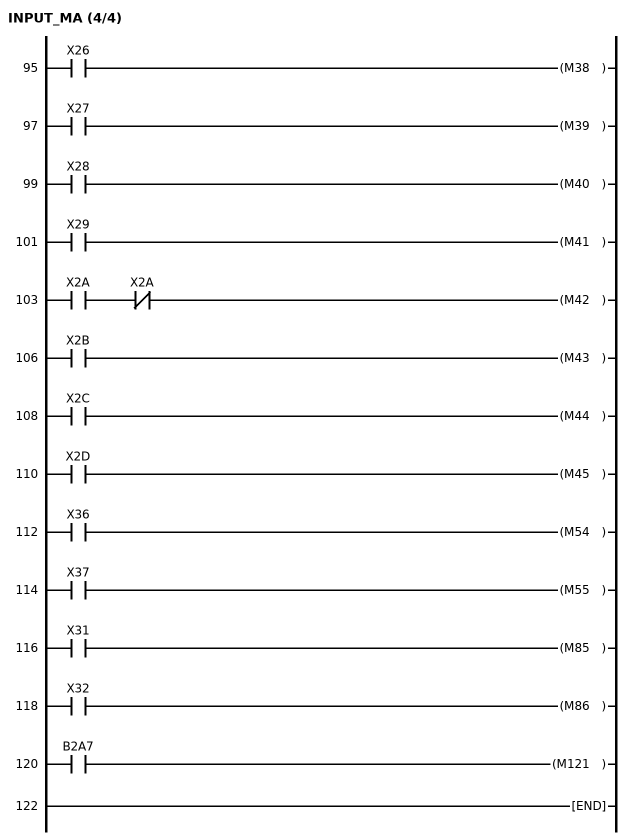
95    LD      X26
      OUT     M38
97    LD      X27
      OUT     M39
99    LD      X28
      OUT     M40
101   LD      X29
      OUT     M41
103   LD      X2A
      ANI     X2A
      OUT     M42
106   LD      X2B
      OUT     M43
108   LD      X2C
      OUT     M44
110   LD      X2D
      OUT     M45
112   LD      X36
      OUT     M54
114   LD      X37
      OUT     M55
116   LD      X31
      OUT     M85
118   LD      X32
      OUT     M86
120   LD      B2A7
      OUT     M121
122   END
END_PROGRAM

PROGRAM MANUAL_P
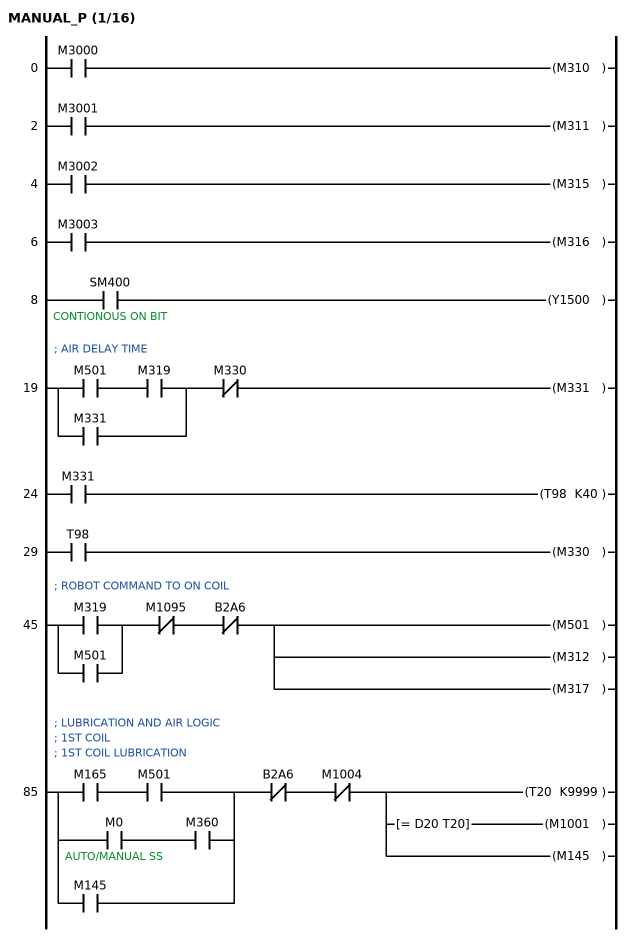
0     LD      M3000
      OUT     M310
2     LD      M3001
      OUT     M311
4     LD      M3002
      OUT     M315
6     LD      M3003
      OUT     M316
8     LD      SM400  ; CONTIONOUS ON BIT
      OUT     Y1500
; AIR DELAY TIME
19    LD      M501
      AND     M319
      OR      M331
      ANI     M330
      OUT     M331
24    LD      M331
      OUT     T98 K40
29    LD      T98
      OUT     M330
; ROBOT COMMAND TO ON COIL
45    LD      M319
      OR      M501
      ANI     M1095
      ANI     B2A6
      OUT     M501
      OUT     M312
      OUT     M317
; LUBRICATION AND AIR LOGIC
; 1ST COIL
; 1ST COIL LUBRICATION
85    LD      M165
      AND     M501
      LD      M0  ; AUTO/MANUAL SS
      AND     M360
      ORB
      OR      M145
      ANI     B2A6
      ANI     M1004
      OUT     T20 K9999
      MPS
      AND=    D20 T20
      OUT     M1001
      MPP
      OUT     M145
